FUNCTION_BLOCK FB_TOR_Spd EXTENDS FB_TOR_Base
//////////////////
//  Smoke and Fire detection system with Typhoon triggering system. 
//////////////////
VAR_INPUT PERSISTENT
	// Parameters of the Object (instance/model specific) 
	ParamTempoEs :TIME:=T#5S;//  (s)Tempo before raising an alarm
END_VAR

VAR_OUTPUT
	//Child objects
	
END_VAR

VAR_INPUT
	// I/O Inputs 		                                     				
		
	
END_VAR

VAR
	//M_ALARMMANAGEMENT VARIABLES//
		FB_PermAlarm				: SR ;					// (NA) FB to maintain Fire Alarm even if sensor stop detection (burn) .
		TON_ES						: TON ; 
 
	//M_STATEMANAGER VARIABLES//
		MesDataExd			: TOR_Standard ;  

		
END_VAR

METHOD M_Execute
//////////////////
//  Method Calls 
/////////////////

VAR 
	// Method local variables (reinitialized at each cycle) 

END_VAR

	
	IF ParamNbSensors = 9 THEN // Use of contactor bi-stable No and NC
		IN_MesState2_IO := NOT IN_MesState2_IO;
	END_IF
SUPER^.M_Execute() ;
END_METHOD

END_FUNCTION_BLOCK

(* stored: Version 1.1.0.1, ProductVersion 3.1.4024.6
   POU FB_TOR_Spd: Id {4070a0da-f099-4f6d-a887-426694246e79}, SpecialFunc None
   Method M_Execute: Id {0bfe5525-c54a-49d9-86f4-8fc08a1d5065} *)
